PROGRAM LDD
VAR
	Start: BOOL:= TRUE;
	Heat: BOOL;
	Cool: BOOL;
	Flush: BOOL;
	Chill: BOOL;
	Hold: BOOL;
	Con1: BOOL;
	Run: BOOL;
	SteamIn: BOOL;
	Drain: BOOL;
	Temp: REAL;
	WaterIn: BOOL;
	GlycolIn: BOOL;
	GlycolOut: BOOL;
	FlushTimer: TON;
	Finished: BOOL;
END_VAR
VAR // added by the converter: edge detectors and wires of the graphical bodies
    _w1, _w2, _w3, _w4, _w5, _w6, _w7, _w8, _w9, _w10 : BOOL;
END_VAR

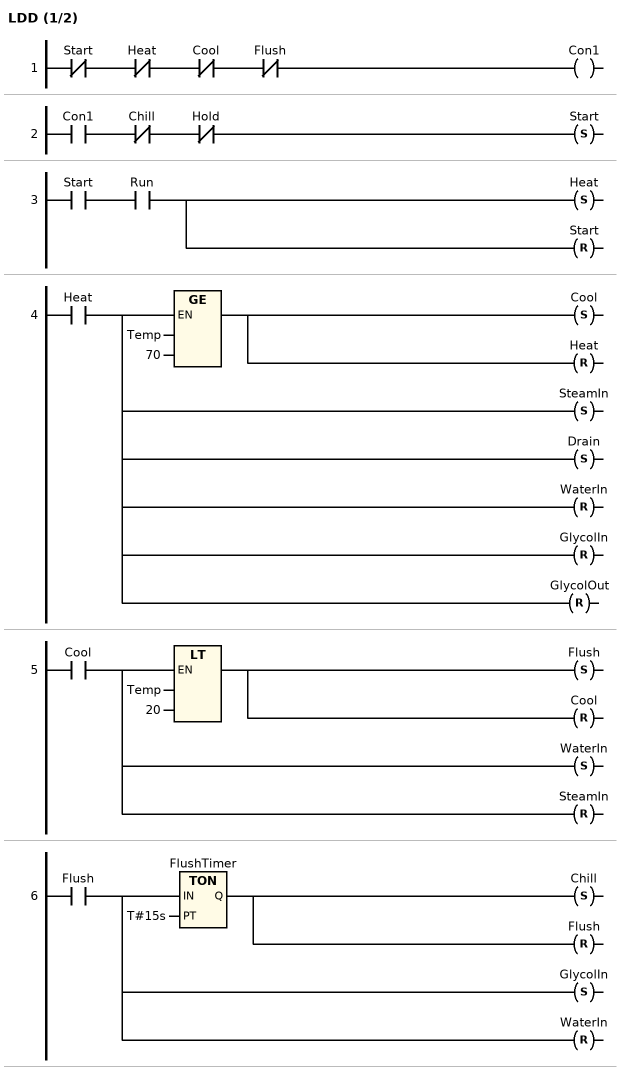
// NETWORK 1
Con1 := NOT Start AND NOT Heat AND NOT Cool AND NOT Flush;

// NETWORK 2
Start S= Con1 AND NOT Chill AND NOT Hold;

// NETWORK 3
_w1 := Start AND Run;
Heat S= _w1;
Start R= _w1;

// NETWORK 4
_w2 := Heat;
_w3 := _w2 AND Temp >= 70;
Cool S= _w3;
Heat R= _w3;
SteamIn S= _w2;
Drain S= _w2;
WaterIn R= _w2;
GlycolIn R= _w2;
GlycolOut R= _w2;

// NETWORK 5
_w4 := Cool;
_w5 := _w4 AND Temp < 20;
Flush S= _w5;
Cool R= _w5;
WaterIn S= _w4;
SteamIn R= _w4;

// NETWORK 6
_w6 := Flush;
FlushTimer(IN := _w6, PT := T#15s); // TON
Chill S= FlushTimer.Q;
Flush R= FlushTimer.Q;
GlycolIn S= _w6;
WaterIn R= _w6;

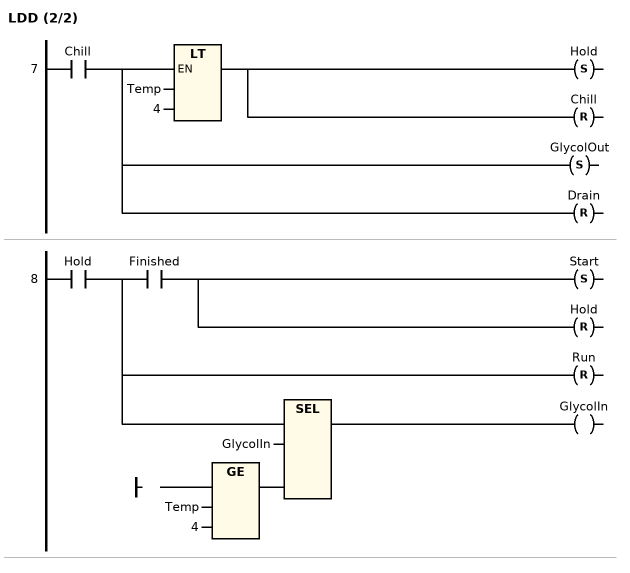
// NETWORK 7
_w7 := Chill;
_w8 := _w7 AND Temp < 4;
Hold S= _w8;
Chill R= _w8;
GlycolOut S= _w7;
Drain R= _w7;

// NETWORK 8
_w9 := Hold;
_w10 := _w9 AND Finished;
Start S= _w10;
Hold R= _w10;
Run R= _w9;
GlycolIn := SEL(_w9, GlycolIn, Temp >= 4);

END_PROGRAM

(* stored: Version 1.1.0.1, ProductVersion 3.1.4024.12
   POU LDD: Id {685dc796-73e5-454c-8f83-0bac94f7fd17}, SpecialFunc None *)
